PROGRAM SetSiemensControlModes
VAR
	i_BessMode		:INT;
	i_InvMode		:INT;
	b_Overule		: BOOL;
	TON_StorageModePulseTrigger: TON ;
	
	b_RobertTest	:BOOL;
	
	Testmode		: INT;
	
	

END_VAR

i_BessMode := InProfinetSiemens.i_BessMode;
i_InvMode  := InProfinetSiemens.i_InvMode;
IF NOT GVL.b_SiemensOverule THEN
	GVL.Gl_ShutdownIntitiatedVisu := FALSE;
	GVL.GL_UserStopVisu := FALSE;
	Safety.b_EmergencyStopVisu := FALSE;
END_IF

CASE i_BessMode OF 
	0:	//REMAIN AT CURRENT MODE
		GVL.b_ActivateSettings := FALSE;
		GVL.GL_ActivateSelectedMode := FALSE;

	1:	//SHUTDOWN
		GVL.Gl_ShutdownIntitiatedVisu := TRUE;
		
		IF (GVL.GL_StorageModeActivate OR GVL.GL_TransportModeActivate) THEN
			GVL.GL_StorageModeButtonPushed := FALSE;
		END_IF
		
	2:	// STORAGE MODE ON
		
		GVL.GL_StorageModeButtonPushed := TRUE;		;
	
		IF DigitalOutputs.b_StorageModeRelay OR GVL.GL_TransportModeActivate THEN
			OutProfinetSIEMENS.i_BessModeFB := 1;
		END_IF
		
		
		
	3: 	// TRANSPORT MODE
		//Integrated in current storage mode.
	
	4: 	// EXT CONTROL MODE
		//TO BE DONE
		
	5:	// Microgrid Mode
		GVL.GL_StorageModeButtonPushed := FALSE;
		IF (NOT DigitalInputs.b_TransferSwitchIOFF OR NOT DigitalInputs.b_TransferSwitchIIOFF) THEN
			GVL.GL_MicroGridModeButtonPushed := TRUE;
			GVL.b_ActivateSettings := TRUE;
			GVL.GL_ActivateSelectedMode := TRUE;
		END_IF
		
	6: // AFE Mode
		//TO BE DONE
		
	7: // ERROR
	Safety.b_EmergencyStopVisu	:=TRUE;
	
	IF safety.b_EmergencyStopSoftwareOK = FALSE THEN
		OutProfinetSIEMENS.i_BessModeFB := 6;
	END_IF
		
END_CASE

CASE i_InvMode	OF
	0: //REMAIN AT CURRENT MODE
	
	1: // INVERTER RUN DISABLE / OFF
		IF GVL.Gl_ShutdownIntitiatedVisu := TRUE THEN
			GVL.GL_UserStopVisu := FALSE;
		ELSE
			GVL.GL_UserStopVisu := TRUE;
		END_IF	
	
		IF GVL.Gl_ModeChangePossible := 1 THEN;
			OutProfinetSIEMENS.i_InvModeFB := 0;
		END_IF
		
	2: // ISOCHRONIOUS MODE
		GVL.i_StartPowerMode := 3;
		GVL.i_StartVoltageMode:= 2;
		
		//WHEN INVERTER MODULATION IS STOPPED, BUT MCCB STILL IN.
		IF NOT GVL.b_InverterRunning AND GVL.b_InverterReadyToOperate THEN  
			GVL.GL_ActivateSelectedMode := TRUE;
		END_IF
		
		
	3: // DROOP MODE (island)
		GVL.i_StartPowerMode := 2;
		GVL.i_StartVoltageMode:= 1;
		
		//WHEN INVERTER MODULATION IS STOPPED, BUT MCCB STILL IN.
		IF NOT GVL.b_InverterRunning AND GVL.b_InverterReadyToOperate THEN  
			GVL.GL_ActivateSelectedMode := TRUE;
		END_IF
		
	
END_CASE

//FEEDBACK SIGNAL BESS MODE
IF safety.b_EmergencyStopSoftwareOK = FALSE THEN
	OutProfinetSIEMENS.i_BessModeFB := 6;
ELSIF GVL.by_Status_ModeSequence = 17 OR GVL.by_Status_ModeSequence = 20 THEN //17 Mode off, 20 Client Setting Active
	OutProfinetSIEMENS.i_BessModeFB := 0;
ELSIF GVL.GL_StorageModeActivate THEN
	OutProfinetSIEMENS.i_BessModeFB := 1;
ELSIF GVL.b_MicroGridModeActive THEN;
	OutProfinetSIEMENS.i_BessModeFB := 4;
END_IF

// ERROR SET TO SIEMENS
IF Diagnostics.b_Error = TRUE THEN
	OutProfinetSIEMENS.i_BessModeFB := 6;
	OutProfinetSIEMENS.i_InvModeFB := 0;
END_IF


//FEEDBACK SIGNAL INVERTER MODE
IF OutProfinetInverter.i_StartPowerMode = 3 AND OutProfinetInverter.i_StartVoltageMode = 2 THEN
		OutProfinetSIEMENS.i_InvModeFB := 1;
ELSIF OutProfinetInverter.i_StartPowerMode = 2 AND OutProfinetInverter.i_StartVoltageMode = 1 THEN
		OutProfinetSIEMENS.i_InvModeFB := 2;
END_IF

END_PROGRAM

(* stored: Version 1.1.0.1, ProductVersion 3.1.4024.12
   POU SetSiemensControlModes: Id {9d616345-4145-42cf-8fd5-93bfa151c796}, SpecialFunc None *)
